(* PLC project io_on_off_valve, Dassault Systèmes ControlBuild 2024x *)
(* stored: creationDateTime 2023-10-03T11:12:49-01:00 *)

PROGRAM panel
  VAR_OUTPUT
    closeValvePB : BOOL := false;
    openValvePB : BOOL := false;
  END_VAR

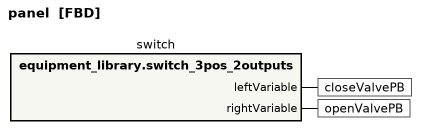
(* FBD diagram, written out as Structured Text *)
switch();
closeValvePB := switch.leftVariable;
openValvePB := switch.rightVariable;
END_PROGRAM

(* Integrated object C/C+OP of an on/off valve *)
PROGRAM io_library.io_on_off_valve
  VAR_INPUT
    acknowledgePB : BOOL := false;
  END_VAR
  VAR_INPUT
    autoMode : BOOL := false;
    manualMode : BOOL := false;
  END_VAR
  VAR_INPUT
    autoCloseCmd : BOOL := false;
    autoOpenCmd : BOOL := false;
  END_VAR
  VAR_INPUT
    inputFlow : REAL := 0.0;
  END_VAR
  VAR_OUTPUT
    openedSensor : BOOL := false;
    closedSensor : BOOL := false;
  END_VAR
  VAR_OUTPUT
    generalFault : BOOL := false;
    outputFlow : REAL := 0.0;
    percentOpening : REAL := 0.0;
  END_VAR

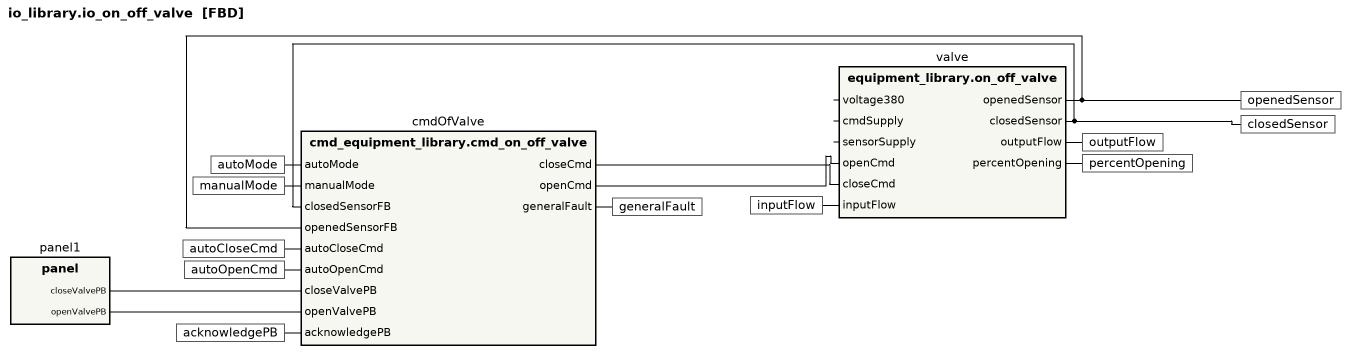
(* FBD diagram, written out as Structured Text *)
panel1();
cmdOfValve(autoMode := autoMode, manualMode := manualMode, closedSensorFB := valve.closedSensor, openedSensorFB := valve.openedSensor, autoCloseCmd := autoCloseCmd, autoOpenCmd := autoOpenCmd, closeValvePB := panel1.closeValvePB, openValvePB := panel1.openValvePB, acknowledgePB := acknowledgePB);
valve(openCmd := cmdOfValve.openCmd, closeCmd := cmdOfValve.closeCmd, inputFlow := inputFlow);
openedSensor := valve.openedSensor;
closedSensor := valve.closedSensor;
outputFlow := valve.outputFlow;
percentOpening := valve.percentOpening;
generalFault := cmdOfValve.generalFault;
END_PROGRAM
